// TIA Portal V20 export
TYPE "LBP_typeConfigData"
TITLE = Configuration parameter / Paramètre de configuration
// User data type for block LBP_ConfigData [DB7] / Type de données utilisateur pour bloc LBP_ConfigData [DB7]
   STRUCT
      MCPNum : Int;   // Inputs starting here / Début des entrées
      MCP1In : Struct   // Pointer / Pointeur
         DBNo : Word;
         Addr : DWord;
      END_STRUCT;
      MCP1Out : Struct   // Pointer / Pointeur
         DBNo : Word;
         Addr : DWord;
      END_STRUCT;
      reservedByte14_25 : Array[14..25] of Byte;
      MCP1BusAdr : Int := 6;
      MCP1Timeout : S5Time := S5T#700MS;
      reservedByte30_31 : Array[30..31] of Byte;
      MCP2In : Struct   // Pointer / Pointeur
         DBNo : Word;
         Addr : DWord;
      END_STRUCT;
      MCP2Out : Struct   // Pointer / Pointeur
         DBNo : Word;
         Addr : DWord;
      END_STRUCT;
      reservedByte44_55 : Array[44..55] of Byte;
      MCP2BusAdr : Int;
      MCP2Timeout : S5Time := S5T#700MS;
      reservedByte60_61 : Array[60..61] of Byte;
      reservedBool62_0 : Bool;
      MCP1Stop : Bool;
      MCP2Stop : Bool;
      MCP1NotSend : Bool;
      MCP2NotSend : Bool;
      reservedBool62_5 : Bool;
      reservedBool62_6 : Bool;
      MCPBusType : Byte := BYTE#16#05;
      HTIf : Int;
      HTIn : Struct   // Pointer / Pointeur
         DBNo : Word;
         Addr : DWord;
      END_STRUCT;
      HTOut : Struct   // Pointer / Pointeur
         DBNo : Word;
         Addr : DWord;
      END_STRUCT;
      reservedByte78_95 : Array[78..95] of Byte;
      HTAdr : Int := 2;
      reservedByte98_107 : Array[98..107] of Byte;
      reservedBool108_0 : Bool;
      HTStop : Bool;
      HTNotSend : Bool;
      NCCyclTimeout : S5Time := S5T#200MS;
      NCRunupTimeout : S5Time := S5T#50S;
      ListMDecGrp : Int;
      reservedBool116_0 : Bool;
      MMCToIF : Bool := TRUE;
      HWheelMMC : Bool := TRUE;
      reservedBool116_3 : Bool;
      MCP_IF_TCS : Bool;
      ExtendChanAxMsg : Bool;
      HMIAxisSel : Bool;
      DeactivateCtrlEnergy : Bool;
      MsgUser : Int := 10;
      reservedBool120_0 : Bool;
      IRAuxfuT : Bool;
      IRAuxfuH : Bool;
      IRAuxfuE : Bool;
      UserVersion : Struct   // Pointer / Pointeur
         DBNo : Word;
         Addr : DWord;
      END_STRUCT;
      OpKeyNum : Int;
      Op1KeyIn : Struct   // Pointer / Pointeur
         DBNo : Word;
         Addr : DWord;
      END_STRUCT;
      Op1KeyOut : Struct   // Pointer / Pointeur
         DBNo : Word;
         Addr : DWord;
      END_STRUCT;
      Op1KeyBusAdr : Int;
      Op2KeyIn : Struct   // Pointer / Pointeur
         DBNo : Word;
         Addr : DWord;
      END_STRUCT;
      Op2KeyOut : Struct   // Pointer / Pointeur
         DBNo : Word;
         Addr : DWord;
      END_STRUCT;
      Op2KeyBusAdr : Int;
      Op1KeyStop : Bool;
      Op2KeyStop : Bool;
      Op1KeyNotSend : Bool;
      Op2KeyNotSend : Bool;
      reservedByte159 : Byte;
      IdentMcpBusAdr : Int;
      IdentMcpProfilNo : Byte;
      IdentMcpBusType : Byte := BYTE#16#05;
      IdentMcpStrobe : Bool;
      MaxModeGroup : Int;   // Outputs starting here / Début des sorties
      MaxChan : Int;
      MaxAxis : Int;
      ActiveChan : Array[1..10] of Bool;
      ActiveAxis : Array[1..31] of Bool;
      MaxNumUserDataInt : Int;
      MaxNumUserDataHex : Int;
      MaxNumUserDataReal : Int;
      IdentMcpType : Byte;
      IdentMcpLengthIn : Byte;
      IdentMcpLengthOut : Byte;
      reservedByte188_199 : Array[188..199] of Byte;   // Static starting here / Début statique
      LBPVersionInfo : String[44];
      UserVersionInfo : String[44];
      GenerateAlarmMsgs : Struct
         NumActAlarmMsgs : UInt;
         Error : Bool;
         StatusID : UInt;
         Status : Word;
      END_STRUCT;
      OpUnitCommId : UInt := 1;   // ID for OpUnitComm / ID pour OpUnitComm
      OpUnitInterfaceId : HW_ANY := 262;   // Hardware identifier of Ethernet interface for OpUnitComm / Identifiant matériel de l'interface Ethernet pour OpUnitComm
      MCP1ConnectionId : CONN_OUC := 1001;   // Connection identifier for MCP 1 / Identifiant de connexion pour MCP 1
      MCP2ConnectionId : CONN_OUC := 1002;   // Connection identifier for MCP 2 / Identifiant de connexion pour MCP 2
      HTConnectionId : CONN_OUC := 1003;   // Connection identifier for handheld unit / Identifiant de connexion pour terminal portatif
      Op1KeyConnectionId : CONN_OUC := 1004;   // Connection identifier for Direct Key 1 / Identifiant de connexion pour Direct Key 1
      Op2KeyConnectionId : CONN_OUC := 1005;   // Connection identifier for Direct Key 2 / Identifiant de connexion pour Direct Key 2
      IdentConnectionId : CONN_OUC := 1006;   // Connection identifier for identification / Identifiant de connexion pour identification
      MCP1LocalUdpPort : UInt := 16001;   // Local UDP port for MCP 1 / Port UDP local pour MCP 1
      MCP2LocalUdpPort : UInt := 16002;   // Local UDP port for MCP 2 / Port UDP local pour MCP 2
      HTLocalUdpPort : UInt := 16003;   // Local UDP port for handheld unit / Port UDP local pour unité de commande portable
      Op1KeyLocalUdpPort : UInt := 16004;   // Local UDP port for Direct Key 1 / Port UDP local pour Direct Key 1
      Op2KeyLocalUdpPort : UInt := 16005;   // Local UDP port for Direct Key 2 / Port UDP local pour Direct Key 2
      IdentLocalUdpPort : UInt := 16006;   // Local UDP port for Ident / Port UDP local pour Ident
      MCP1Error : Bool;   // Error MCP 1 / Erreur MCP 1
      MCP1Status : Word;   // Error information MCP 1 / Information erreur MCP 1
      MCP2Error : Bool;   // Error MCP 2 / Erreur MCP 2
      MCP2Status : Word;   // Error information MCP 2 / Information erreur MCP 2
      HTError : Bool;   // Error handheld unit / Erreur terminal portatif
      HTStatus : Word;   // Error information handheld unit / Information erreur terminal portatif
      Op1KeyError : Bool;   // Error Direct Key 1 / Erreur Direct Key 1
      Op1KeyStatus : Word;   // Error information Direct Key 1 / Information erreur Direct Key 1
      Op2KeyError : Bool;   // Error Direct Key 2 / Erreur Direct Key 2
      Op2KeyStatus : Word;   // Error information Direct Key 2 / Information erreur Direct Key 2
      IdentError : Bool;   // Error identification / Identification d'erreur
      IdentStatus : Word;   // Error information Identification / Identification d'erreur Identification
      MCP1Ready : Bool;   // MCP1 connected / MCP1 connecté
      MCP2Ready : Bool;   // MCP2 connected / MCP2 connecté
      HTReady : Bool;   // Handheld unit connected / Terminal portatif connecté
      Op1KeyReady : Bool;   // Direct Key 1 connected / Direct Key 1 connecté
      Op2KeyReady : Bool;   // Direct Key 2 connected / Direct Key 2 connecté
   END_STRUCT;
END_TYPE
